FUNCTION_BLOCK SystemTest
VAR_INPUT
END_VAR
VAR_OUTPUT
END_VAR
VAR
END_VAR

IF IO.g_ReadIO THEN
	IO.g_ReadIO := FALSE;
ELSE
	IO.g_ReadIO := TRUE;
END_IF

END_FUNCTION_BLOCK

(* stored: Version 1.1.0.1, ProductVersion 3.1.4024.6
   POU SystemTest: Id {62fb5ba1-c269-41db-82c7-d3069fec3701}, SpecialFunc None *)
